INTERFACE I_SINT EXTENDS I_Datatype

{warning disable C5410}
PROPERTY PUBLIC Value : REFERENCE TO SINT
{warning restore C5410}
GET
END_GET
END_PROPERTY

END_INTERFACE

(* stored: Version 1.1.0.1, ProductVersion 3.1.4024.15
   Itf I_SINT: Id {af8d9b79-b3d6-0fe5-2487-8054253ef912}
   Property Value: Id {4e9574dc-ac84-0283-2957-89519c13c6a5}
   Get Get: Id {be1daa36-d78f-0cae-2900-174e85da11d7} *)
